// TIA Portal project "brama_V17" (V17)

(* hardware
DEVICE "S7-1200 station_1"  S7-1200 Station
   slot 0: "Rack_0"  Rack  V1.0
   slot 1: "PLC_1"  CPU 1212C AC/DC/Rly  6ES7 212-1BD30-0XB0  V2.2
   slot 101: "CM 1241 (RS232)_1"  6ES7 241-1AH30-0XB0  V1.0
*)

// ===== PLC "PLC_1"  CPU 1212C AC/DC/Rly =====

VAR_GLOBAL   // PLC tag table "Default tag table"
   "Tag_1" AT %I0.0 : Bool;
   "Tag_2" AT %I0.1 : Bool;
   "Tag_3" AT %I0.2 : Bool;
   "Tag_4" AT %Q0.1 : Bool;
   "Tag_5" AT %Q0.2 : Bool;
   "Tag_6" AT %Q0.4 : Bool;
   "Tag_7" AT %Q0.3 : Bool;
   "Tag_8" AT %Q0.5 : Bool;
   "Tag_9" AT %M50.0 : Bool;
   "Tag_10" AT %Q0.0 : Bool;
   "Clock_Byte" AT %MB0 : Byte;
   "Clock_10Hz" AT %M0.0 : Bool;
   "Clock_5Hz" AT %M0.1 : Bool;
   "Clock_2.5Hz" AT %M0.2 : Bool;
   "Clock_2Hz" AT %M0.3 : Bool;
   "Clock_1.25Hz" AT %M0.4 : Bool;
   "Clock_1Hz" AT %M0.5 : Bool;
   "Clock_0.625Hz" AT %M0.6 : Bool;
   "Clock_0.5Hz" AT %M0.7 : Bool;
END_VAR

DATA_BLOCK "BramaFun_DB"   // DB16
{ S7_Optimized_Access := 'TRUE' }
VERSION : 0.1
// stored: InstanceOfName BramaFun
"BramaFun"
BEGIN
END_DATA_BLOCK

// folder: System blocks/Program resources

DATA_BLOCK "IEC_Timer_0_DB"   // DB1
{ S7_Optimized_Access := 'TRUE' }
AUTHOR : Simatic
FAMILY : IEC
NAME : IEC_TMR
VERSION : 1.0
// stored: InstanceOfName IEC_TIMER
"IEC_TIMER"
BEGIN
END_DATA_BLOCK

DATA_BLOCK "IEC_Timer_0_DB_1"   // DB2
{ S7_Optimized_Access := 'TRUE' }
AUTHOR : Simatic
FAMILY : IEC
NAME : IEC_TMR
VERSION : 1.0
// stored: InstanceOfName IEC_TIMER
"IEC_TIMER"
BEGIN
END_DATA_BLOCK

DATA_BLOCK "IEC_Timer_0_DB_2"   // DB3
{ S7_Optimized_Access := 'TRUE' }
AUTHOR : Simatic
FAMILY : IEC
NAME : IEC_TMR
VERSION : 1.0
// stored: InstanceOfName IEC_TIMER
"IEC_TIMER"
BEGIN
END_DATA_BLOCK

DATA_BLOCK "IEC_Timer_0_DB_3"   // DB4
{ S7_Optimized_Access := 'TRUE' }
AUTHOR : Simatic
FAMILY : IEC
NAME : IEC_TMR
VERSION : 1.0
// stored: InstanceOfName IEC_TIMER
"IEC_TIMER"
BEGIN
END_DATA_BLOCK

DATA_BLOCK "IEC_Timer_0_DB_4"   // DB6
{ S7_Optimized_Access := 'TRUE' }
AUTHOR : Simatic
FAMILY : IEC
NAME : IEC_TMR
VERSION : 1.0
// stored: InstanceOfName IEC_TIMER
"IEC_TIMER"
BEGIN
END_DATA_BLOCK

DATA_BLOCK "IEC_Timer_0_DB_5"   // DB7
{ S7_Optimized_Access := 'TRUE' }
AUTHOR : Simatic
FAMILY : IEC
NAME : IEC_TMR
VERSION : 1.0
// stored: InstanceOfName IEC_TIMER
"IEC_TIMER"
BEGIN
END_DATA_BLOCK

DATA_BLOCK "IEC_Timer_0_DB_6"   // DB8
{ S7_Optimized_Access := 'TRUE' }
AUTHOR : Simatic
FAMILY : IEC
NAME : IEC_TMR
VERSION : 1.0
// stored: InstanceOfName IEC_TIMER
"IEC_TIMER"
BEGIN
END_DATA_BLOCK

DATA_BLOCK "IEC_Counter_0_DB"   // DB9
{ S7_Optimized_Access := 'TRUE' }
AUTHOR : Simatic
FAMILY : IEC
NAME : CNTR
VERSION : 1.0
// stored: InstanceOfName IEC_COUNTER
"IEC_COUNTER"
BEGIN
END_DATA_BLOCK

DATA_BLOCK "IEC_Timer_0_DB_7"   // DB10
{ S7_Optimized_Access := 'TRUE' }
AUTHOR : Simatic
FAMILY : IEC
NAME : IEC_TMR
VERSION : 1.0
// stored: InstanceOfName IEC_TIMER
"IEC_TIMER"
BEGIN
END_DATA_BLOCK

DATA_BLOCK "IEC_Timer_0_DB_8"   // DB11
{ S7_Optimized_Access := 'TRUE' }
AUTHOR : Simatic
FAMILY : IEC
NAME : IEC_TMR
VERSION : 1.0
// stored: InstanceOfName IEC_TIMER
"IEC_TIMER"
BEGIN
END_DATA_BLOCK

DATA_BLOCK "IEC_Timer_0_DB_9"   // DB12
{ S7_Optimized_Access := 'TRUE' }
AUTHOR : Simatic
FAMILY : IEC
NAME : IEC_TMR
VERSION : 1.0
// stored: InstanceOfName IEC_TIMER
"IEC_TIMER"
BEGIN
END_DATA_BLOCK

DATA_BLOCK "IEC_Timer_0_DB_10"   // DB13
{ S7_Optimized_Access := 'TRUE' }
AUTHOR : Simatic
FAMILY : IEC
NAME : IEC_TMR
VERSION : 1.0
// stored: InstanceOfName IEC_TIMER
"IEC_TIMER"
BEGIN
END_DATA_BLOCK

DATA_BLOCK "IEC_Timer_0_DB_11"   // DB14
{ S7_Optimized_Access := 'TRUE' }
AUTHOR : Simatic
FAMILY : IEC
NAME : IEC_TMR
VERSION : 1.0
// stored: InstanceOfName IEC_TIMER
"IEC_TIMER"
BEGIN
END_DATA_BLOCK

DATA_BLOCK "IEC_Timer_0_DB_12"   // DB15
{ S7_Optimized_Access := 'TRUE' }
AUTHOR : Simatic
FAMILY : IEC
NAME : IEC_TMR
VERSION : 1.0
// stored: InstanceOfName IEC_TIMER
"IEC_TIMER"
BEGIN
END_DATA_BLOCK

DATA_BLOCK "IEC_Timer_0_DB_13"   // DB17
{ S7_Optimized_Access := 'TRUE' }
AUTHOR : Simatic
FAMILY : IEC
NAME : IEC_TMR
VERSION : 1.0
// stored: InstanceOfName IEC_TIMER
"IEC_TIMER"
BEGIN
END_DATA_BLOCK

DATA_BLOCK "IEC_Counter_0_DB_1"   // DB18
{ S7_Optimized_Access := 'TRUE' }
AUTHOR : Simatic
FAMILY : IEC
NAME : CNTR
VERSION : 1.0
// stored: InstanceOfName IEC_COUNTER
"IEC_COUNTER"
BEGIN
END_DATA_BLOCK

DATA_BLOCK "IEC_Timer_0_DB_14"   // DB19
{ S7_Optimized_Access := 'TRUE' }
AUTHOR : Simatic
FAMILY : IEC
NAME : IEC_TMR
VERSION : 1.0
// stored: InstanceOfName IEC_TIMER
"IEC_TIMER"
BEGIN
END_DATA_BLOCK

DATA_BLOCK "IEC_Timer_0_DB_15"   // DB20
{ S7_Optimized_Access := 'TRUE' }
AUTHOR : Simatic
FAMILY : IEC
NAME : IEC_TMR
VERSION : 1.0
// stored: InstanceOfName IEC_TIMER
"IEC_TIMER"
BEGIN
END_DATA_BLOCK

DATA_BLOCK "IEC_Timer_0_DB_16"   // DB21
{ S7_Optimized_Access := 'TRUE' }
AUTHOR : Simatic
FAMILY : IEC
NAME : IEC_TMR
VERSION : 1.0
// stored: InstanceOfName IEC_TIMER
"IEC_TIMER"
BEGIN
END_DATA_BLOCK

DATA_BLOCK "IEC_Timer_0_DB_17"   // DB22
{ S7_Optimized_Access := 'TRUE' }
AUTHOR : Simatic
FAMILY : IEC
NAME : IEC_TMR
VERSION : 1.0
// stored: InstanceOfName IEC_TIMER
"IEC_TIMER"
BEGIN
END_DATA_BLOCK

DATA_BLOCK "IEC_Timer_0_DB_18"   // DB23
{ S7_Optimized_Access := 'TRUE' }
AUTHOR : Simatic
FAMILY : IEC
NAME : IEC_TMR
VERSION : 1.0
// stored: InstanceOfName IEC_TIMER
"IEC_TIMER"
BEGIN
END_DATA_BLOCK

// folder: (top level)

FUNCTION_BLOCK "BramaFun"   // FB2, LAD
{ S7_Optimized_Access := 'TRUE' }
VERSION : 0.1
   VAR_INPUT
      przycisk : Bool;
      foto1 : Bool;
      foto2 : Bool;
      clock : Bool;
   END_VAR
   VAR_OUTPUT
      lampa : Bool;
   END_VAR
   VAR_IN_OUT
      silnik2_open : Bool;
      silnik1_open : Bool;
      silnik1_close : Bool;
      silnik2_close : Bool;
   END_VAR
   VAR
      open : Bool;   // potwierdzenie - brama otwarta
      close : Bool := 1;   // potwierdzenie - brama zamknieta
      stan_bramy : USInt;   // 0 - nic, 1 - otwieranie, 2 - zamykanie
      przycisk_zbocze : Bool;
      silnik2_open_zbocze : Bool;
      silnik1_close_zbocze : Bool;
      TON_out : Bool;
      TON_out_zbocze : Bool;
   END_VAR
   VAR_TEMP   // added for the SCL form of the ladder/FBD networks
      _w1 : Bool;
      _w2 : Bool;
      _w3 : Bool;
   END_VAR
BEGIN

REGION Network 1: uruchomienie otwierania/zamykania
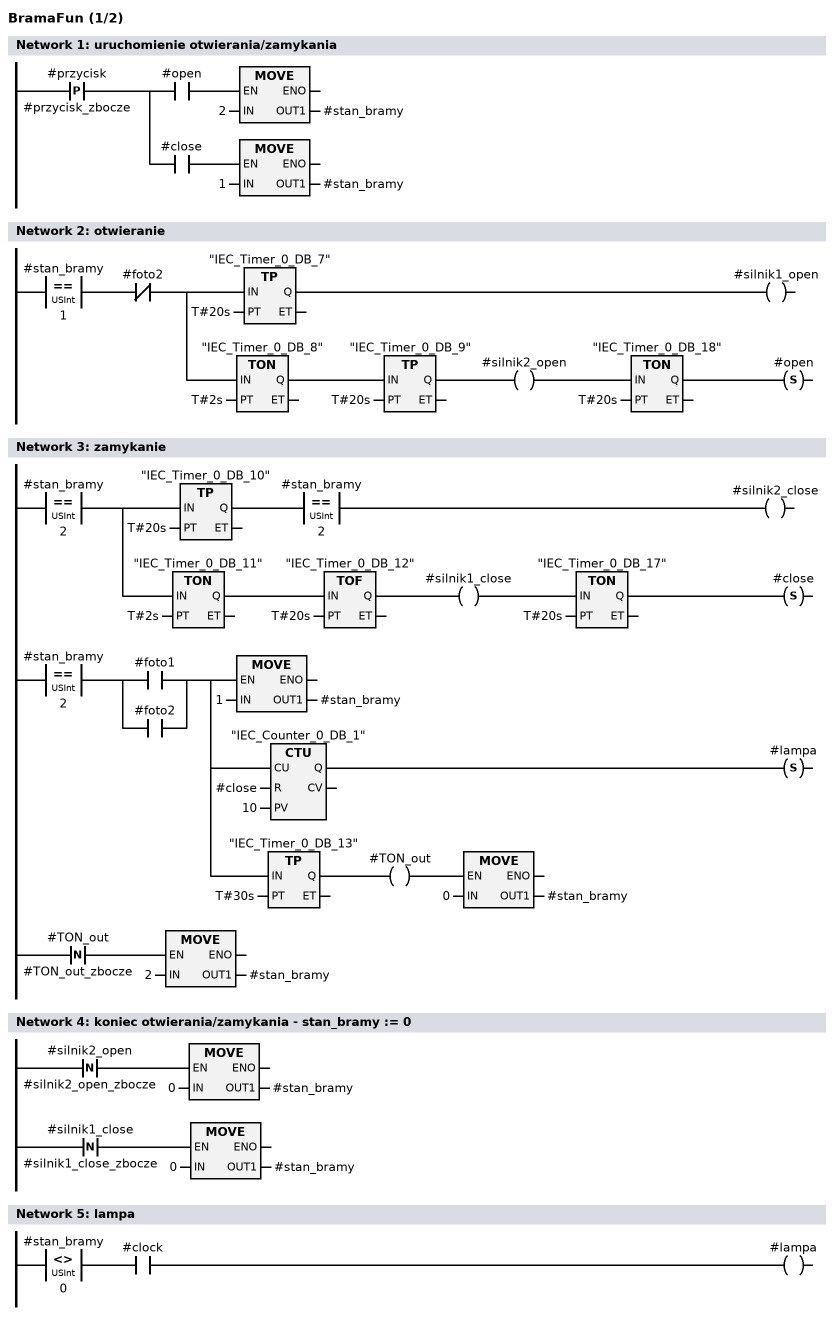
   RUNG wire#powerrail
      P_Contact(operand := #przycisk, bit := #przycisk_zbocze)
      wire#w1
      Contact( #open )
      { S7_GenerateENO := "TRUE" } Move(in := 2, out1 => #stan_bramy)
   END_RUNG
   RUNG wire#w1
      Contact( #close )
      { S7_GenerateENO := "TRUE" } Move(in := 1, out1 => #stan_bramy)
   END_RUNG
   // the same network as SCL:
   #_w1 := #przycisk AND NOT #przycisk_zbocze;   // rising edge of #przycisk
   #przycisk_zbocze := #przycisk;
   IF #_w1 AND #open THEN #stan_bramy := 2; END_IF;
   IF #_w1 AND #close THEN #stan_bramy := 1; END_IF;
END_REGION

REGION Network 2: otwieranie
   #_w1 := (#stan_bramy = 1) AND NOT #foto2;
   "IEC_Timer_0_DB_7".TP(IN := #_w1, PT := T#20s);
   #silnik1_open := "IEC_Timer_0_DB_7".Q;
   "IEC_Timer_0_DB_8".TON(IN := #_w1, PT := T#2s);
   "IEC_Timer_0_DB_9".TP(IN := "IEC_Timer_0_DB_8".Q, PT := T#20s);
   #silnik2_open := "IEC_Timer_0_DB_9".Q;
   "IEC_Timer_0_DB_18".TON(IN := "IEC_Timer_0_DB_9".Q, PT := T#20s);
   IF "IEC_Timer_0_DB_18".Q THEN #open := TRUE; END_IF;
END_REGION

REGION Network 3: zamykanie
   #_w1 := #stan_bramy = 2;
   "IEC_Timer_0_DB_10".TP(IN := #_w1, PT := T#20s);
   #silnik2_close := "IEC_Timer_0_DB_10".Q AND (#stan_bramy = 2);
   "IEC_Timer_0_DB_11".TON(IN := #_w1, PT := T#2s);
   "IEC_Timer_0_DB_12".TOF(IN := "IEC_Timer_0_DB_11".Q, PT := T#20s);
   #silnik1_close := "IEC_Timer_0_DB_12".Q;
   "IEC_Timer_0_DB_17".TON(IN := "IEC_Timer_0_DB_12".Q, PT := T#20s);
   IF "IEC_Timer_0_DB_17".Q THEN #close := TRUE; END_IF;
   #_w2 := (#stan_bramy = 2) AND (#foto1 OR #foto2);
   IF #_w2 THEN #stan_bramy := 1; END_IF;
   "IEC_Counter_0_DB_1".CTU(CU := #_w2, R := #close, PV := 10);
   IF "IEC_Counter_0_DB_1".Q THEN #lampa := TRUE; END_IF;
   "IEC_Timer_0_DB_13".TP(IN := #_w2, PT := T#30s);
   #TON_out := "IEC_Timer_0_DB_13".Q;
   IF "IEC_Timer_0_DB_13".Q THEN #stan_bramy := 0; END_IF;
   #_w3 := NOT #TON_out AND #TON_out_zbocze;   // falling edge of #TON_out
   #TON_out_zbocze := #TON_out;
   IF #_w3 THEN #stan_bramy := 2; END_IF;
END_REGION

REGION Network 4: koniec otwierania/zamykania - stan_bramy := 0
   RUNG wire#powerrail
      N_Contact(operand := #silnik2_open, bit := #silnik2_open_zbocze)
      { S7_GenerateENO := "TRUE" } Move(in := 0, out1 => #stan_bramy)
   END_RUNG
   RUNG wire#powerrail
      N_Contact(operand := #silnik1_close, bit := #silnik1_close_zbocze)
      { S7_GenerateENO := "TRUE" } Move(in := 0, out1 => #stan_bramy)
   END_RUNG
   // the same network as SCL:
   #_w1 := NOT #silnik2_open AND #silnik2_open_zbocze;   // falling edge of #silnik2_open
   #silnik2_open_zbocze := #silnik2_open;
   IF #_w1 THEN #stan_bramy := 0; END_IF;
   #_w2 := NOT #silnik1_close AND #silnik1_close_zbocze;   // falling edge of #silnik1_close
   #silnik1_close_zbocze := #silnik1_close;
   IF #_w2 THEN #stan_bramy := 0; END_IF;
END_REGION

REGION Network 5: lampa
   RUNG wire#powerrail
      { S7_Templates := "SrcType := USInt" } NE_Contact(in1 := #stan_bramy, in2 := 0)
      Contact( #clock )
      Coil( #lampa )
   END_RUNG
   // the same network as SCL:
   #lampa := (#stan_bramy <> 0) AND #clock;
END_REGION

REGION Network 6: gdy chodzi silnik => brama nie jest ani w pelni otwarta, ani w pelni zamknieta
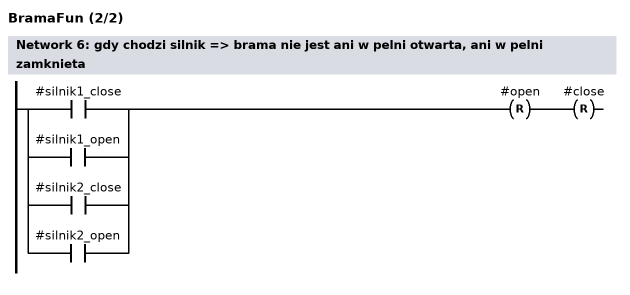
   RUNG wire#powerrail
      Contact( #silnik1_close )
      wire#w1
      R_Coil( #open )
      R_Coil( #close )
   END_RUNG
   RUNG wire#powerrail
      Contact( #silnik1_open )
   END_RUNG wire#w1
   RUNG wire#powerrail
      Contact( #silnik2_close )
   END_RUNG wire#w1
   RUNG wire#powerrail
      Contact( #silnik2_open )
   END_RUNG wire#w1
   // the same network as SCL:
   IF #silnik1_close OR #silnik1_open OR #silnik2_close OR #silnik2_open THEN
       #open := FALSE;
       #close := FALSE;
   END_IF;
END_REGION
END_FUNCTION_BLOCK

ORGANIZATION_BLOCK "Main"   // OB1, LAD, ProgramCycle
TITLE = "Main Program Sweep (Cycle)"
{ S7_Optimized_Access := 'TRUE' }
VERSION : 0.1
BEGIN

REGION Network 1
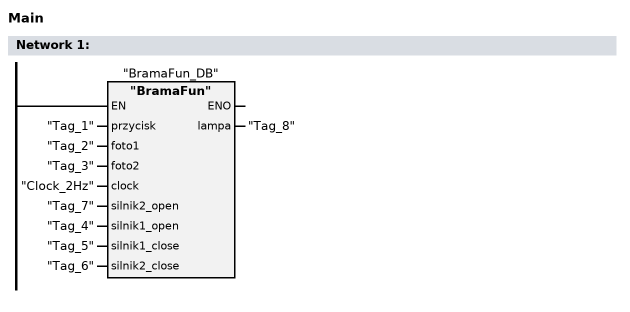
   RUNG wire#powerrail
      "BramaFun_DB"(przycisk := "Tag_1", foto1 := "Tag_2", foto2 := "Tag_3", clock := "Clock_2Hz", silnik2_open := "Tag_7", silnik1_open := "Tag_4", silnik1_close := "Tag_5", silnik2_close := "Tag_6", lampa => "Tag_8")
   END_RUNG
   // the same network as SCL:
   "BramaFun_DB"(przycisk := "Tag_1",   // "BramaFun"
                 foto1 := "Tag_2",
                 foto2 := "Tag_3",
                 clock := "Clock_2Hz",
                 silnik2_open := "Tag_7",
                 silnik1_open := "Tag_4",
                 silnik1_close := "Tag_5",
                 silnik2_close := "Tag_6",
                 lampa => "Tag_8");
END_REGION
END_ORGANIZATION_BLOCK